//----------------------------------------------------------------------------//
//            Copyright 2018 Rieckermann Engineering Operations               //
//                Automatically Generated File - Do Not Edit                  //
//----------------------------------------------------------------------------//
// Description:                                                               //
// This file defines the Control Recipe structure.                            //
//----------------------------------------------------------------------------//
// Revision history:                                                          //
// Rev By               Date        CC        Note                            //
// 1.0 David Paspa      21-May-2018 NA        Reboot for S7-1500.             //
//----------------------------------------------------------------------------//
DATA_BLOCK "dbRECIPE"
TITLE = Control Recipe
{ S7_Optimized_Access := 'FALSE' }
AUTHOR : REO
NAME : dbRECIPE
VERSION : 1.0

@@TEMPLATE_BEGIN|createClassNone@@
STRUCT
    isMaster : Bool := @@MASTERRECIPE@@;
    recipeInfo : Struct
        rcpPCMXNumber : Int;
        rcpPCMXDataRecordNumber : Int;
        rcpPCMXStatus : Int;
        rcpPCSYNumber : Int;
        rcpPCSYDataRecordNumber : Int;
        rcpPCSYStatus : Int;
    END_STRUCT;
    recipeMaster : Struct
@@ATTR_BEGIN|RECIPE_PARAMETER_CLASS@@
        PC@@CLASS@@ : Struct
@@ATTR_BEGIN|RECIPE_PARAMETERS@@
            @@BLOCKPARAMETER@@ : @@PARAMETERDATATYPE@@;      // @@PARAMETERDESCRIPTION@@
@@ATTR_END|RECIPE_PARAMETERS@@
        END_STRUCT;
@@ATTR_END|RECIPE_PARAMETER_CLASS@@
    END_STRUCT;
    recipeControl : Struct
@@ATTR_BEGIN|RECIPE_PARAMETER_CLASS@@
@@ATTR_BEGIN|getInstancesForClass@@
        PC@@INSTANCE@@ : Struct
@@ATTR_BEGIN|RECIPE_PARAMETERS@@
            @@BLOCKPARAMETER@@ : @@PARAMETERDATATYPE@@;      // @@PARAMETERDESCRIPTION@@
@@ATTR_END|RECIPE_PARAMETERS@@
        END_STRUCT;
@@ATTR_END|getInstancesForClass@@
@@ATTR_END|RECIPE_PARAMETER_CLASS@@
    END_STRUCT;
END_STRUCT;
@@TEMPLATE_END@@

BEGIN
END_DATA_BLOCK
